// TIA Portal V17 export
// export: Created 2025-01-08T13:55:35.1133155Z, ExportSetting WithDefaults, DisplayName Totally Integrated Automation Portal, DisplayVersion V17, DisplayName TIA Portal Openness, DisplayVersion V17, DisplayName TIA Portal Version Control Interface, DisplayVersion V17, DisplayName SINAMICS Startdrive Advanced, DisplayVersion V17 Update2, DisplayName SINAMICS Startdrive G130, G150, S120, S150, SINAMICS MV, S210, DisplayVersion V17 Update2, DisplayName SINAMICS Startdrive G110M, G120, G120C, G120D, G120P, G115D, DisplayVersion V17 Update2, DisplayName STEP 7 Professional, DisplayVersion V17, DisplayName STEP 7 Safety, DisplayVersion V17, DisplayName WinCC Advanced, DisplayVersion V17
DATA_BLOCK "DB - Settings_From_PC"   // DB63
{ S7_Optimized_Access := 'FALSE' }
VERSION : 0.1
// stored: AutoNumber true, DBAccessibleFromOPCUA true, DBAccessibleFromWebserver true, IsOnlyStoredInLoadMemory false, IsWriteProtectedInAS false
   VAR RETAIN
      DispenseLabelSensorCalibration : LReal := 200.0;   // Avstånd från Gap givare till tunga
      SpeedDifferenceDispenser : LReal := -5.0;   // Hastighetsskillnad Dispensering
      DispenseLabelDistance : LReal := -610.0;   // Etikettlängd
      IndexWheel_HomingDistance : LReal := -510.0;   // Indexhjul homing avstånd
      SpeedDifferenceDispeningSplice : LReal := 0.0;   // Hastighetsskillnad Dispensering Start
      PercentageToChangeLabelPosition : LReal := 1.0;   // Procent att ändra etikettposition
      NumberOfRejectsToIgnore : LReal := 20.0;   // Antal underkända dosor att ignorera
      NumberOfProductsBeforeAdjustStart : LReal := 4.0;   // Antal dosor innan justering vid start
      NumberOfProductsBeforeAdjustStop : LReal := 5.0;   // Antal dosor innan justering
      RotateProductMPerMinToDegreesPerSecondCalibrationValue : LReal := 48.0;   // Rotera product motor kalibreringsvärde
      SideRejectDelay : LReal := 0.0;   // Banderoll reject fördröjning
      OrientationValue : LReal := 0.0;   // Orienteringsmotorer kalibrerings värde
      OrientaionCorrectionValue : LReal := 0.0;   // Orintering korrigeringsvärde
      SideSyncLength : LReal;
   END_VAR
BEGIN
END_DATA_BLOCK
